// TIA Portal project "Hydraulikaggregat" (V15)

(* hardware
DEVICE "S7-1200-Station_1"  S7-1200 Station
   slot 0: "Baugruppenträger_0"  S7-1200 Rack  Rack  V1.0
   slot 1: "PLC_1"  CPU 1214C DC/DC/Rly  6ES7 214-1HG40-0XB0  V4.2
DEVICE "HMI_1"  KTP700 Basic PN
   slot 0: "HMI_1"  KTP700 Basic PN  6AV2 123-2GB03-0AX0  15.0.0.0
   slot 1: "HMI_RT_1"  KTP700 Basic PN  6AV2 123-2GB03-0AX0  15.0.0.0
   slot 5: "HMI_1.IE_CP_1"  PROFINET Interface  15.0.0.0
      slot 1: "PROFINET Schnittstelle_1"  PROFINET Interface
         slot 1: "Port_1"  Port
*)

// ===== PLC "PLC_1"  CPU 1214C DC/DC/Rly =====

VAR_GLOBAL   // PLC tag table "Standard-Variablentabelle"
   "Clock_Byte" AT %MB100 : Byte;
   "Clock_10Hz" AT %M100.0 : Bool;
   "Clock_5Hz" AT %M100.1 : Bool;
   "Clock_2.5Hz" AT %M100.2 : Bool;
   "Clock_2Hz" AT %M100.3 : Bool;
   "Clock_1.25Hz" AT %M100.4 : Bool;
   "Clock_1Hz" AT %M100.5 : Bool;
   "Clock_0.625Hz" AT %M100.6 : Bool;
   "Clock_0.5Hz" AT %M100.7 : Bool;
   "S1" AT %I0.0 : Bool;   // Anlage Start
   "S2" AT %I0.1 : Bool;   // Anlage Stop
   "S3" AT %I0.2 : Bool;   // Störung Quittieren
   "B1" AT %I0.3 : Bool;   // Füllstand in Ordnung
   "B2" AT %I0.4 : Bool;   // Füllstand Mitte
   "B3" AT %I0.5 : Bool;   // Füllstand Überdruck
   "F5" AT %I0.6 : Bool;   // Motorschutzschalter
   "P1" AT %Q0.0 : Bool;   // Störung Motor
   "P2" AT %Q0.1 : Bool;   // Überdruck
   "P3" AT %Q0.2 : Bool;   // Druck erreicht
   "P4" AT %Q0.3 : Bool;   // Ölstand min.
   "Q1" AT %Q0.4 : Bool;   // Netzschütz
   "Q2" AT %Q0.5 : Bool;   // Sternschütz
   "Q3" AT %Q0.6 : Bool;   // Dreieckschütz
   "Merker Sammelstörung" AT %M0.0 : Bool;
   "Merker Anlage Betriebsbereit" AT %M0.1 : Bool;
   "Merker Ölstand min." AT %M0.2 : Bool;
END_VAR

DATA_BLOCK "HMI"   // DB3
{ S7_Optimized_Access := 'TRUE' }
VERSION : 0.1
   VAR
      "Hydraulik Start" : Bool;
      "Hydraulik Stop" : Bool;
   END_VAR
BEGIN
END_DATA_BLOCK

// folder: System blocks/Program resources

DATA_BLOCK "IEC_Timer_0_DB"   // DB1
{ S7_Optimized_Access := 'TRUE' }
AUTHOR : Simatic
FAMILY : IEC
NAME : IEC_TMR
VERSION : 1.0
// stored: InstanceOfName IEC_TIMER
"IEC_TIMER"
BEGIN
END_DATA_BLOCK

DATA_BLOCK "IEC_Timer_0_DB_1"   // DB2
{ S7_Optimized_Access := 'TRUE' }
AUTHOR : Simatic
FAMILY : IEC
NAME : IEC_TMR
VERSION : 1.0
// stored: InstanceOfName IEC_TIMER
"IEC_TIMER"
BEGIN
END_DATA_BLOCK

// folder: (top level)

FUNCTION "Hydraulikaggregat" : Void   // FC1, FBD
TITLE = Hydraulikaggregat
{ S7_Optimized_Access := 'TRUE' }
VERSION : 0.1
BEGIN

REGION Network 1: Anlage Start
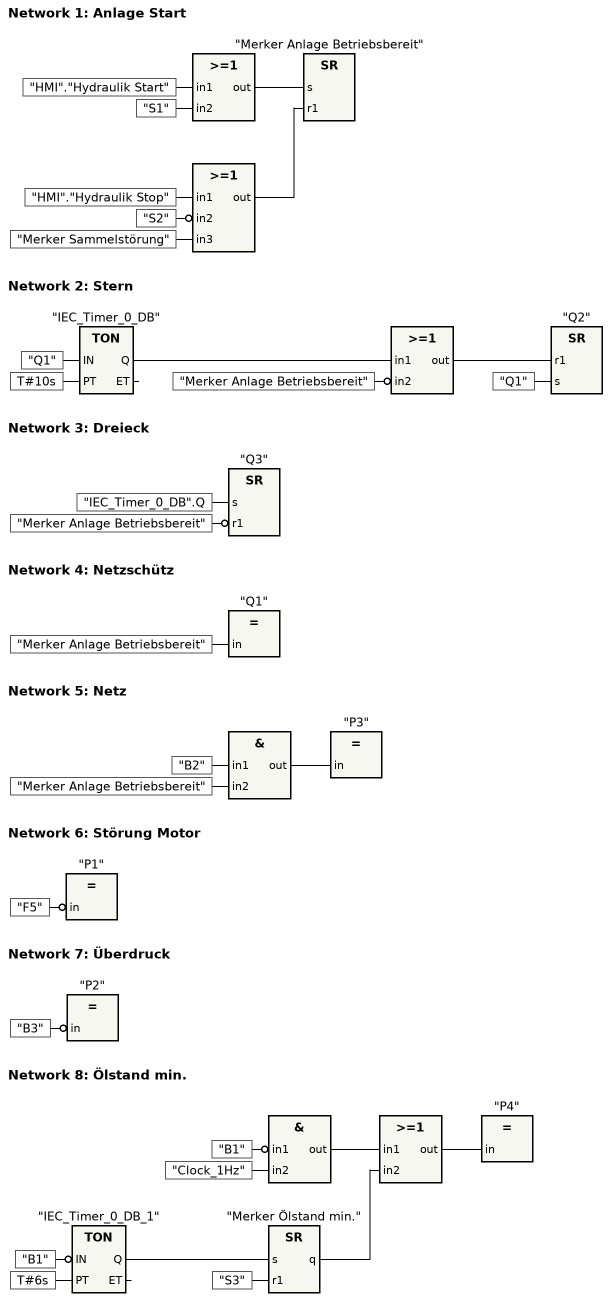
   IF "HMI"."Hydraulik Start" OR "S1" THEN
       "Merker Anlage Betriebsbereit" := TRUE;   // SR flip-flop
   END_IF;
   IF "HMI"."Hydraulik Stop" OR NOT "S2" OR "Merker Sammelstörung" THEN
       "Merker Anlage Betriebsbereit" := FALSE;
   END_IF;
END_REGION

REGION Network 2: Stern
   "IEC_Timer_0_DB".TON(IN := "Q1", PT := T#10s);
   IF "Q1" THEN
       "Q2" := TRUE;   // SR flip-flop
   END_IF;
   IF "IEC_Timer_0_DB".Q OR NOT "Merker Anlage Betriebsbereit" THEN "Q2" := FALSE; END_IF;
END_REGION

REGION Network 3: Dreieck
   IF "IEC_Timer_0_DB".Q THEN
       "Q3" := TRUE;   // SR flip-flop
   END_IF;
   IF NOT "Merker Anlage Betriebsbereit" THEN "Q3" := FALSE; END_IF;
END_REGION

REGION Network 4: Netzschütz
   "Q1" := "Merker Anlage Betriebsbereit";
END_REGION

REGION Network 5: Netz
   "P3" := "B2" AND "Merker Anlage Betriebsbereit";
END_REGION

REGION Network 6: Störung Motor
   "P1" := NOT "F5";
END_REGION

REGION Network 7: Überdruck
   "P2" := NOT "B3";
END_REGION

REGION Network 8: Ölstand min.
   "IEC_Timer_0_DB_1".TON(IN := NOT "B1", PT := T#6s);
   IF "IEC_Timer_0_DB_1".Q THEN
       "Merker Ölstand min." := TRUE;   // SR flip-flop
   END_IF;
   IF "S3" THEN "Merker Ölstand min." := FALSE; END_IF;
   "P4" := (NOT "B1" AND "Clock_1Hz") OR "Merker Ölstand min.";
END_REGION

REGION Network 9: Sammelstörung
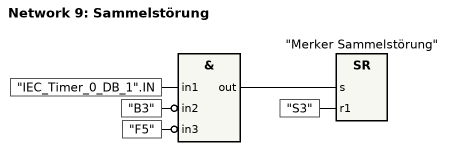
   IF "IEC_Timer_0_DB_1".IN AND NOT "B3" AND NOT "F5" THEN
       "Merker Sammelstörung" := TRUE;   // SR flip-flop
   END_IF;
   IF "S3" THEN "Merker Sammelstörung" := FALSE; END_IF;
END_REGION
END_FUNCTION

ORGANIZATION_BLOCK "Main"   // OB1, LAD, ProgramCycle
TITLE = "Main Program Sweep (Cycle)"
{ S7_Optimized_Access := 'TRUE' }
VERSION : 0.1
   VAR_INPUT
      Initial_Call : Bool;   // Initial call of this OB
      Remanence : Bool;   // =True, if remanent data are available
   END_VAR
BEGIN

REGION Network 1
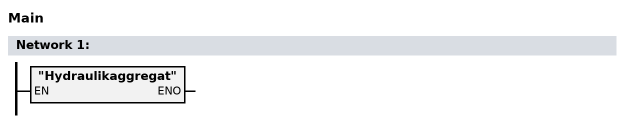
   RUNG wire#powerrail
      "Hydraulikaggregat"()
   END_RUNG
   // the same network as SCL:
   "Hydraulikaggregat"();
END_REGION
END_ORGANIZATION_BLOCK

(* ===== HMI "HMI_RT_1" =====
system functions are stored by id; their names below are inferred from use
connection "HMI_Verbindung_1": ETHERNET, SMART_S7_1200_OMS

HMI tags "Standard-Variablentabelle"
   "P3" : Bool = PLC P3 AT %Q0.2, 100 ms
   "P1" : Bool = PLC P1 AT %Q0.0, 100 ms
   "P4" : Bool = PLC P4 AT %Q0.3, 100 ms
   "P2" : Bool = PLC P2 AT %Q0.1, 100 ms
   "HMI_Hydraulik Start" : Bool = PLC HMI."Hydraulik Start", 1 s
   "HMI_Hydraulik Stop" : Bool = PLC HMI."Hydraulik Stop", 1 s

screen "Bild_1" 800x480
   Button "Schaltfläche_1" at 55,147 size 200x84; TextOff 'Hyrdaulik Start'
      on Press: function_b14e0dd5("HMI_Hydraulik Start", 0)
   Circle "Kreis_1" at 540,97 size 50x50
      Appearance <- "P3"
   Button "Schaltfläche_2" at 55,284 size 200x84; TextOff 'Hyrdaulik Stop'
      on Press: function_b14e0dd5("HMI_Hydraulik Stop", 0)
   Circle "Kreis_2" at 540,174 size 50x50
      Appearance <- "P1"
   Circle "Kreis_3" at 540,251 size 50x50
      Appearance <- "P2"
   Circle "Kreis_4" at 540,334 size 50x50
      Appearance <- "P4"
   TextField "Textfeld_1" at 55,14 size 233x23; Text 'Hydraulikaggregat Standart'
   TextField "Textfeld_3" at 59,46 size 309x23; Text 'Prüflingsnummer 007, am 20.06.2020'
   TextField "Textfeld_2" at 599,345 size 147x23; Text 'Ölstand minimum'
   TextField "Textfeld_4" at 599,261 size 158x23; Text 'Störung Überdruck'
   TextField "Textfeld_5" at 599,187 size 122x23; Text 'Störung Motor'
   TextField "Textfeld_6" at 599,108 size 121x23; Text 'Druck erreicht'
*)